Universal Robots PolyScope program: Simran_CNC_Program_FINAL.urp

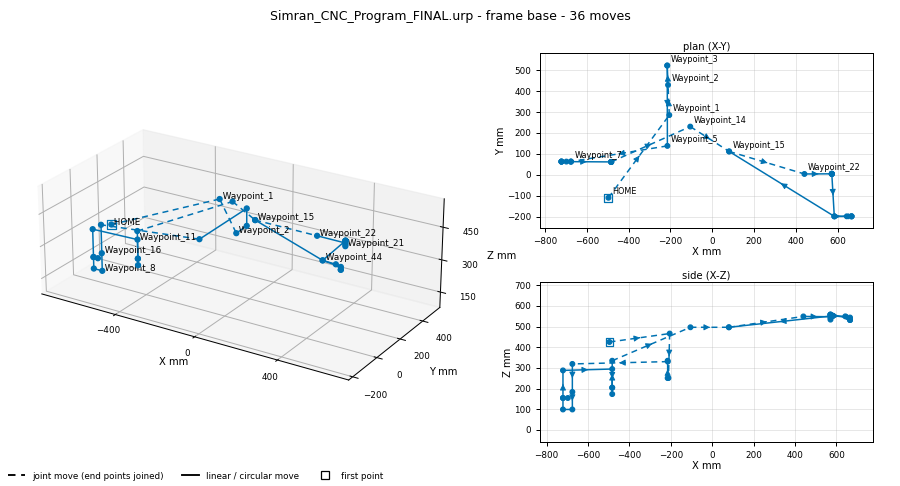
[picture p0: tool path of Simran_CNC_Program_FINAL.urp in frame base, 36 of 36 moves have a stored position in this frame; points joined in program order, loops and branches not executed]
Program Simran_CNC_Program_FINAL (createdIn=3.4.3.361 lastSavedIn=3.4.3.361 directory=/programs installation=default robotSerialNumber=2016352713)
Calibrated DH parameters: a=[0.000153, -0.131035, -0.301404, -0.000338, 0.000464, 0]; d=[0.089115, 288.344324, 295.555383, -583.78943, 0.09474, 0.082313]; alpha=[1.57022, 0.001403, 0.00043, 1.569471, -1.569661, 0]; deltaTheta=[-0.000066, 1.257544, -0.563043, -0.694494, -0.000004, 0.000038]
Robot Program (runOnlyOnce=true motionType=MoveJ speed=1.047198 acceleration=1.396263 useActiveTCP=false)
  MoveJ speed 60 deg/s, acceleration 80 deg/s^2 (useActiveTCP=false)
    Waypoint HOME: TCP in base x=-496.442 y=-110.074 z=425.318 mm, rx=1.2792 ry=2.857 rz=0.0029 rad; joints [-0.001, -88.582, 89.405, -90.126, -89.769, -41.695] deg
    Call Tool_OPEN
  'TURN TOWARDS CONVEYOR'
  MoveJ speed 60 deg/s, acceleration 80 deg/s^2 (useActiveTCP=false)
    Waypoint Waypoint_1: TCP in base x=-205.447 y=285.381 z=466.125 mm, rx=-1.2263 ry=-2.8909 rz=-0.0134 rad; joints [-72.357, -110.466, 101.648, -81.546, -90.206, -116.353] deg
  'PICK UP RAW MATERIALS BIN'
  MoveJ speed 60 deg/s, acceleration 80 deg/s^2 (useActiveTCP=false)
    Waypoint Waypoint_2: TCP in base x=-211.365 y=429.379 z=251.173 mm, rx=1.2208 ry=2.8789 rz=0.0239 rad; joints [-76.836, -86.876, 114.31, -117.592, -91.124, -120.798] deg
  MoveL speed 250 mm/s, acceleration 1200 mm/s^2 (useActiveTCP=false) feature=Base
    Waypoint Waypoint_3: TCP in base x=-215.251 y=522.375 z=251.019 mm, rx=1.2191 ry=2.8755 rz=0.0088 rad; joints [-78.664, -75.619, 100.862, -114.845, -90.993, -122.619] deg
    Waypoint Waypoint_4: motionParameters(jointSpeed=1.047198 jointAcceleration=1.396263 cartesianSpeed=0.02 cartesianAcceleration=0.02); TCP in base x=-215.258 y=522.371 z=334.743 mm, rx=1.2191 ry=2.8754 rz=0.0087 rad; joints [-78.665, -79.363, 92.558, -102.798, -90.989, -122.628] deg
    Waypoint Waypoint_5: TCP in base x=-214.547 y=138.032 z=330.506 mm, rx=1.2327 ry=2.8739 rz=0.0237 rad; joints [-57.762, -126.871, 129.262, -92.139, -91.154, -101.3] deg
  'PLACE RAW MATERIALS BIN'
  MoveJ speed 60 deg/s, acceleration 80 deg/s^2 (useActiveTCP=false)
    SuppressedNode
      Waypoint Waypoint_6: TCP in base x=-214.554 y=138.064 z=330.528 mm, rx=2.3465 ry=2.0595 rz=0.0117 rad; joints [-57.965, -126.737, 129.007, -91.172, -90.574, -50.482] deg
    Waypoint Waypoint_7: TCP in base x=-675.818 y=62.939 z=319.323 mm, rx=-2.9058 ry=-1.1583 rz=0.0302 rad; joints [-14.657, -63.822, 74.31, -101.769, -89.898, 31.98] deg
  MoveL speed 250 mm/s, acceleration 1200 mm/s^2 (useActiveTCP=false) feature=Base
    Waypoint Waypoint_16: TCP in base x=-675.802 y=62.877 z=183.922 mm, rx=-2.8969 ry=-1.1806 rz=0.0305 rad; joints [-14.658, -57.697, 85.778, -119.362, -89.886, 31.113] deg
    Waypoint Waypoint_8: motionParameters(jointSpeed=1.047198 jointAcceleration=1.396263 cartesianSpeed=0.02 cartesianAcceleration=0.02); TCP in base x=-675.776 y=62.901 z=99.21 mm, rx=-2.8958 ry=-1.1834 rz=0.0305 rad; joints [-14.66, -51.451, 89.635, -129.469, -89.886, 31.01] deg
    Waypoint Waypoint_9: TCP in base x=-721.173 y=62.9 z=99.19 mm, rx=-2.8958 ry=-1.1834 rz=0.0306 rad; joints [-13.746, -46.438, 80.218, -125.063, -89.908, 31.929] deg
    Waypoint Waypoint_10: motionParameters(jointSpeed=1.047198 jointAcceleration=1.396263 cartesianSpeed=0.25 cartesianAcceleration=1.2); TCP in base x=-721.174 y=62.931 z=154.677 mm, rx=-2.8958 ry=-1.1834 rz=0.0306 rad; joints [-13.745, -50.326, 77.932, -118.89, -89.901, 31.925] deg
    Waypoint Waypoint_17: motionParameters(jointSpeed=1.047198 jointAcceleration=1.396263 cartesianSpeed=0.02 cartesianAcceleration=0.02); TCP in base x=-697.665 y=62.978 z=154.655 mm, rx=-2.8959 ry=-1.1833 rz=0.0304 rad; joints [-14.203, -53.165, 82.942, -121.061, -89.89, 31.463] deg; flange x=-697.689 y=62.9 z=154.695 mm, rx=-2.8958 ry=-1.1834 rz=0.0306 rad
    Waypoint Waypoint_10: motionParameters(jointSpeed=1.047198 jointAcceleration=1.396263 cartesianSpeed=0.25 cartesianAcceleration=1.2); TCP in base x=-721.174 y=62.931 z=154.677 mm, rx=-2.8958 ry=-1.1834 rz=0.0306 rad; joints [-13.745, -50.326, 77.932, -118.89, -89.901, 31.925] deg
    Waypoint Waypoint_18: TCP in base x=-721.163 y=62.916 z=288.004 mm, rx=-2.8958 ry=-1.1834 rz=0.0304 rad; joints [-13.747, -56.577, 67.748, -102.456, -89.893, 31.91] deg; flange x=-721.174 y=62.931 z=288.056 mm, rx=-2.8958 ry=-1.1834 rz=0.0306 rad
  'PICK UP 1ST BLOCK'
  MoveL speed 250 mm/s, acceleration 1200 mm/s^2 (useActiveTCP=false) feature=Base
    Waypoint Waypoint_11: TCP in base x=-483.165 y=61.413 z=294.634 mm, rx=-2.894 ry=-1.1612 rz=-0.0146 rad; joints [-20.032, -88.315, 108.927, -111.051, -91.293, 26.31] deg; flange x=-483.17 y=61.41 z=294.731 mm, rx=-2.8939 ry=-1.1611 rz=-0.0143 rad
    Waypoint Waypoint_12: TCP in base x=-483.165 y=61.376 z=204.49 mm, rx=-2.8937 ry=-1.1612 rz=-0.0142 rad; joints [-20.033, -82.152, 117.078, -125.366, -91.297, 26.319] deg; flange x=-483.17 y=61.41 z=204.448 mm, rx=-2.8939 ry=-1.1611 rz=-0.0143 rad
    Waypoint Waypoint_23: motionParameters(jointSpeed=1.047198 jointAcceleration=1.396263 cartesianSpeed=0.02 cartesianAcceleration=0.02); TCP in base x=-483.17 y=61.41 z=173.567 mm, rx=-2.8939 ry=-1.1611 rz=-0.0143 rad; joints [-20.034, -79.281, 119.255, -130.412, -91.296, 26.321] deg
    Wait Sleep waitTime=0.5
    Call Tool_CLOSE
    Wait Sleep waitTime=1
    Waypoint Waypoint_12: motionParameters(jointSpeed=1.047198 jointAcceleration=1.396263 cartesianSpeed=0.02 cartesianAcceleration=0.02); TCP in base x=-483.165 y=61.376 z=204.49 mm, rx=-2.8937 ry=-1.1612 rz=-0.0142 rad; joints [-20.033, -82.152, 117.078, -125.366, -91.297, 26.319] deg; flange x=-483.17 y=61.41 z=204.448 mm, rx=-2.8939 ry=-1.1611 rz=-0.0143 rad
    Waypoint Waypoint_13: TCP in base x=-483.174 y=61.383 z=334.81 mm, rx=-2.894 ry=-1.1612 rz=-0.0146 rad; joints [-20.033, -90.016, 104.509, -104.919, -91.292, 26.304] deg
  MoveJ speed 60 deg/s, acceleration 80 deg/s^2 (useActiveTCP=false)
    Waypoint Waypoint_14: TCP in base x=-105.18 y=230.288 z=496.414 mm, rx=-1.2069 ry=-2.8666 rz=-0.0233 rad; joints [-91.595, -124.024, 103.951, -71.307, -88.599, -135.903] deg
    Waypoint Waypoint_15: TCP in base x=80.805 y=111.483 z=496.435 mm, rx=-1.2494 ry=-2.8485 rz=-0.0239 rad; joints [-180.178, -141.465, 106.176, -53.368, -88.466, -222.831] deg
    Wait Sleep waitTime=0.5
    Set DigitalOutput pin=door; digitalValue=1
    Wait Sleep waitTime=6
  'PLACE 1st BLOCK IN CNC'
  MoveJ speed 60 deg/s, acceleration 80 deg/s^2 (useActiveTCP=false)
    Waypoint Waypoint_22: TCP in base x=440.76 y=3.757 z=548.887 mm, rx=-1.2046 ry=-2.8864 rz=0.0111 rad; joints [-193.886, -95.387, 77.565, -71.268, -90.219, -238.54] deg
  MoveL speed 250 mm/s, acceleration 1200 mm/s^2 (useActiveTCP=false) feature=Base
    SuppressedNode
      Waypoint Waypoint_24: motionParameters(jointSpeed=1.047198 jointAcceleration=1.396263 cartesianSpeed=0.05 cartesianAcceleration=0.02); TCP in base x=551.7 y=-51.289 z=595.114 mm, rx=-2.8876 ry=-1.1713 rz=-0.0332 rad; joints [-197.055, -76.915, 50.59, -63.644, -88.035, -151.148] deg; flange x=551.728 y=-51.253 z=595.093 mm, rx=-2.8876 ry=-1.1713 rz=-0.0331 rad
    Waypoint Waypoint_20: motionParameters(jointSpeed=1.047198 jointAcceleration=1.396263 cartesianSpeed=0.05 cartesianAcceleration=0.025); TCP in base x=571.71 y=4.472 z=547.422 mm, rx=-1.2202 ry=-2.8799 rz=0.011 rad; joints [-190.617, -76.822, 57.791, -70.042, -90.155, -234.626] deg
    Waypoint Waypoint_21: motionParameters(jointSpeed=1.047198 jointAcceleration=1.396263 cartesianSpeed=0.05 cartesianAcceleration=0.01); TCP in base x=571.707 y=4.437 z=533.436 mm, rx=-1.2201 ry=-2.8798 rz=0.0111 rad; joints [-190.615, -77.492, 60.769, -72.35, -90.155, -234.624] deg; flange x=571.725 y=4.478 z=533.464 mm, rx=-1.2201 ry=-2.8799 rz=0.011 rad
    Call Tool_OPEN
    Wait Sleep waitTime=1
    Waypoint Waypoint_25: motionParameters(jointSpeed=1.047198 jointAcceleration=1.396263 cartesianSpeed=0.1 cartesianAcceleration=0.05); TCP in base x=571.711 y=4.432 z=557.354 mm, rx=-1.2201 ry=-2.8798 rz=0.0112 rad; joints [-190.623, -76.277, 55.552, -68.342, -90.155, -234.628] deg
    Call Tool_CLOSE
    Wait Sleep waitTime=1
    Waypoint Waypoint_26: motionParameters(jointSpeed=1.047198 jointAcceleration=1.396263 cartesianSpeed=0.25 cartesianAcceleration=0.1); TCP in base x=571.669 y=4.458 z=557.394 mm, rx=-0.0745 ry=-3.1304 rz=0.0184 rad; joints [-190.545, -76.378, 55.781, -68.858, -90.687, -277.744] deg; flange x=571.707 y=4.437 z=557.356 mm, rx=-0.0745 ry=-3.1303 rz=0.0184 rad
    SuppressedNode
      Waypoint Waypoint_27: motionParameters(jointSpeed=1.047198 jointAcceleration=1.396263 cartesianSpeed=0.025 cartesianAcceleration=0.01); TCP in base x=571.697 y=4.439 z=548.626 mm, rx=-0.0744 ry=-3.1304 rz=0.0184 rad; joints [-190.544, -76.857, 57.748, -70.346, -90.688, -277.743] deg
    SuppressedNode
      Waypoint Waypoint_26: motionParameters(jointSpeed=1.047198 jointAcceleration=1.396263 cartesianSpeed=0.1 cartesianAcceleration=0.05); TCP in base x=571.669 y=4.458 z=557.394 mm, rx=-0.0745 ry=-3.1304 rz=0.0184 rad; joints [-190.545, -76.378, 55.781, -68.858, -90.687, -277.744] deg; flange x=571.707 y=4.437 z=557.356 mm, rx=-0.0745 ry=-3.1303 rz=0.0184 rad
    Waypoint Waypoint_28: motionParameters(jointSpeed=1.047198 jointAcceleration=1.396263 cartesianSpeed=0.025 cartesianAcceleration=0.01); TCP in base x=571.706 y=4.422 z=540.796 mm, rx=-0.0745 ry=-3.1303 rz=0.0183 rad; joints [-190.543, -77.247, 59.44, -71.648, -90.688, -277.741] deg
    Waypoint Waypoint_26: motionParameters(jointSpeed=1.047198 jointAcceleration=1.396263 cartesianSpeed=0.25 cartesianAcceleration=0.1); TCP in base x=571.669 y=4.458 z=557.394 mm, rx=-0.0745 ry=-3.1304 rz=0.0184 rad; joints [-190.545, -76.378, 55.781, -68.858, -90.687, -277.744] deg; flange x=571.707 y=4.437 z=557.356 mm, rx=-0.0745 ry=-3.1303 rz=0.0184 rad
    Waypoint Waypoint_25: motionParameters(jointSpeed=1.047198 jointAcceleration=1.396263 cartesianSpeed=0.15 cartesianAcceleration=0.1); TCP in base x=571.711 y=4.432 z=557.354 mm, rx=-1.2201 ry=-2.8798 rz=0.0112 rad; joints [-190.623, -76.277, 55.552, -68.342, -90.155, -234.628] deg
    Waypoint Waypoint_44: motionParameters(jointSpeed=1.047198 jointAcceleration=1.396263 cartesianSpeed=0.1 cartesianAcceleration=0.05); TCP in base x=583.705 y=-198.923 z=551.901 mm, rx=-1.2205 ry=-2.8797 rz=0.0114 rad; joints [-209.035, -69.295, 47.056, -66.94, -90.423, -253.024] deg; flange x=583.758 y=-198.858 z=551.858 mm, rx=-1.2202 ry=-2.8797 rz=0.0112 rad
    Waypoint Waypoint_45: motionParameters(jointSpeed=1.047198 jointAcceleration=1.396263 cartesianSpeed=0.025 cartesianAcceleration=0.01); TCP in base x=643.414 y=-198.777 z=549.256 mm, rx=-1.2201 ry=-2.8799 rz=0.0113 rad; joints [-206.542, -58.298, 30.69, -61.552, -90.389, -250.524] deg; flange x=643.446 y=-198.824 z=549.179 mm, rx=-1.2201 ry=-2.8798 rz=0.0112 rad
    Waypoint Waypoint_46: motionParameters(jointSpeed=1.047198 jointAcceleration=1.396263 cartesianSpeed=0.025 cartesianAcceleration=0.01); TCP in base x=666.192 y=-198.791 z=531.433 mm, rx=-1.2198 ry=-2.8799 rz=0.0113 rad; joints [-205.699, -55.151, 28.355, -62.353, -90.381, -249.682] deg; flange x=666.19 y=-198.848 z=531.398 mm, rx=-1.2199 ry=-2.8798 rz=0.0112 rad
    Waypoint Waypoint_47: motionParameters(jointSpeed=1.047198 jointAcceleration=1.396263 cartesianSpeed=0.025 cartesianAcceleration=0.01); TCP in base x=666.173 y=-198.919 z=531.389 mm, rx=1.1834 ry=2.7931 rz=0.0671 rad; joints [-206.093, -58.682, 36.074, -73.343, -87.071, -249.923] deg; flange x=666.19 y=-198.848 z=531.398 mm, rx=1.1833 ry=2.7932 rz=0.0672 rad
    Waypoint Waypoint_48: motionParameters(jointSpeed=1.047198 jointAcceleration=1.396263 cartesianSpeed=0.025 cartesianAcceleration=0.01); TCP in base x=666.164 y=-198.888 z=543.546 mm, rx=-1.22 ry=-2.8797 rz=0.0113 rad; joints [-205.701, -53.361, 23.259, -59.048, -90.382, -249.683] deg
    Waypoint Waypoint_44: motionParameters(jointSpeed=1.047198 jointAcceleration=1.396263 cartesianSpeed=0.05 cartesianAcceleration=0.01); TCP in base x=583.705 y=-198.923 z=551.901 mm, rx=-1.2205 ry=-2.8797 rz=0.0114 rad; joints [-209.035, -69.295, 47.056, -66.94, -90.423, -253.024] deg; flange x=583.758 y=-198.858 z=551.858 mm, rx=-1.2202 ry=-2.8797 rz=0.0112 rad
    Waypoint Waypoint_15: motionParameters(jointSpeed=1.047198 jointAcceleration=1.396263 cartesianSpeed=0.25 cartesianAcceleration=0.1); TCP in base x=80.805 y=111.483 z=496.435 mm, rx=-1.2494 ry=-2.8485 rz=-0.0239 rad; joints [-180.178, -141.465, 106.176, -53.368, -88.466, -222.831] deg
    Wait Sleep waitTime=0.5
    Set DigitalOutput pin=door; digitalValue=0
    Wait Sleep waitTime=6
  'TOP TO BOTTOM'
  SuppressedNode
    MoveL speed 250 mm/s, acceleration 1200 mm/s^2 (useActiveTCP=false) feature=Base
      Set DigitalOutput pin=door; digitalValue=1
      Wait Sleep waitTime=6
      Waypoint Waypoint_22: motionParameters(jointSpeed=1.047198 jointAcceleration=1.396263 cartesianSpeed=0.25 cartesianAcceleration=0.1); TCP in base x=440.76 y=3.757 z=548.887 mm, rx=-1.2046 ry=-2.8864 rz=0.0111 rad; joints [-193.886, -95.387, 77.565, -71.268, -90.219, -238.54] deg
      Waypoint Waypoint_25: motionParameters(jointSpeed=1.047198 jointAcceleration=1.396263 cartesianSpeed=0.05 cartesianAcceleration=0.025); TCP in base x=571.711 y=4.432 z=557.354 mm, rx=-1.2201 ry=-2.8798 rz=0.0112 rad; joints [-190.623, -76.277, 55.552, -68.342, -90.155, -234.628] deg
      Call Tool_OPEN
      Wait Sleep waitTime=1
      Waypoint Waypoint_21: motionParameters(jointSpeed=1.047198 jointAcceleration=1.396263 cartesianSpeed=0.05 cartesianAcceleration=0.01); TCP in base x=571.707 y=4.437 z=533.436 mm, rx=-1.2201 ry=-2.8798 rz=0.0111 rad; joints [-190.615, -77.492, 60.769, -72.35, -90.155, -234.624] deg; flange x=571.725 y=4.478 z=533.464 mm, rx=-1.2201 ry=-2.8799 rz=0.011 rad
      Call Tool_CLOSE
      Wait Sleep waitTime=1
      Waypoint Waypoint_19: TCP in base x=571.698 y=4.439 z=560.42 mm, rx=-1.2202 ry=-2.8799 rz=0.0111 rad; joints [-190.62, -76.099, 54.845, -67.822, -90.153, -234.624] deg
      Waypoint Waypoint_24: TCP in base x=466.899 y=-34.446 z=560.48 mm, rx=-1.2202 ry=-2.8801 rz=0.011 rad; joints [-197.739, -91.133, 71.811, -69.799, -90.261, -241.762] deg
      Waypoint Waypoint_29: TCP in base x=332.54 y=-34.477 z=503.635 mm, rx=0.6252 ry=1.4734 rz=0.6267 rad; joints [-213.592, -111.621, 122.767, -191.492, -56.436, -223.787] deg
      Waypoint Waypoint_30: TCP in base x=413.921 y=-34.5 z=444.937 mm, rx=0.6252 ry=1.4734 rz=0.6267 rad; joints [-205.154, -95.603, 120.061, -204.763, -64.896, -223.835] deg
      Waypoint Waypoint_31: TCP in base x=413.908 y=-34.513 z=404.929 mm, rx=0.6253 ry=1.4734 rz=0.6266 rad; joints [-205.157, -92.629, 123.961, -211.635, -64.899, -223.839] deg
      Call Tool_OPEN
      Wait Sleep waitTime=1
      Waypoint Waypoint_32: motionParameters(jointSpeed=1.047198 jointAcceleration=1.396263 cartesianSpeed=0.05 cartesianAcceleration=0.01); TCP in base x=341.668 y=-34.501 z=404.92 mm, rx=0.6254 ry=1.4734 rz=0.6266 rad; joints [-212.365, -104.17, 133.396, -209.558, -57.68, -223.799] deg
      Waypoint Waypoint_33: motionParameters(jointSpeed=1.047198 jointAcceleration=1.396263 cartesianSpeed=0.05 cartesianAcceleration=0.01); TCP in base x=456.404 y=-34.465 z=589.86 mm, rx=-1.2203 ry=-2.88 rz=0.0107 rad; joints [-198.151, -91.019, 67.08, -65.184, -90.269, -242.178] deg
      Waypoint Waypoint_34: motionParameters(jointSpeed=1.047198 jointAcceleration=1.396263 cartesianSpeed=0.05 cartesianAcceleration=0.01); TCP in base x=565.728 y=-34.472 z=589.874 mm, rx=-1.2204 ry=-2.88 rz=0.0107 rad; joints [-194.649, -74.859, 48.544, -62.786, -90.203, -238.651] deg
      Waypoint Waypoint_35: motionParameters(jointSpeed=1.047198 jointAcceleration=1.396263 cartesianSpeed=0.05 cartesianAcceleration=0.01); TCP in base x=565.729 y=-34.449 z=574.404 mm, rx=-1.2202 ry=-2.88 rz=0.0106 rad; joints [-194.646, -75.994, 52.51, -65.617, -90.203, -238.649] deg
      Call Tool_CLOSE
      Wait Sleep waitTime=1
      Waypoint Waypoint_36: motionParameters(jointSpeed=1.047198 jointAcceleration=1.396263 cartesianSpeed=0.05 cartesianAcceleration=0.01); TCP in base x=565.735 y=-34.443 z=588.812 mm, rx=-1.2203 ry=-2.8801 rz=0.0107 rad; joints [-194.649, -74.944, 48.83, -62.987, -90.203, -238.651] deg
      Waypoint Waypoint_37: motionParameters(jointSpeed=1.047198 jointAcceleration=1.396263 cartesianSpeed=0.05 cartesianAcceleration=0.01); TCP in base x=378.265 y=-34.505 z=598.175 mm, rx=0.6269 ry=1.4775 rz=0.6256 rad; joints [-208.263, -105.692, 104.96, -179.298, -61.758, -223.949] deg
      Waypoint Waypoint_38: motionParameters(jointSpeed=1.047198 jointAcceleration=1.396263 cartesianSpeed=0.05 cartesianAcceleration=0.01); TCP in base x=382.478 y=-34.517 z=408.781 mm, rx=0.627 ry=1.4775 rz=0.6256 rad; joints [-207.853, -97.824, 127.848, -210.054, -62.197, -223.96] deg
      Waypoint Waypoint_39: motionParameters(jointSpeed=1.047198 jointAcceleration=1.396263 cartesianSpeed=0.025 cartesianAcceleration=0.01); TCP in base x=382.46 y=-34.495 z=390.09 mm, rx=0.6169 ry=1.454 rz=0.6313 rad; joints [-207.851, -95.528, 129.464, -215.6, -62.214, -223.196] deg
      Call Tool_OPEN
      Wait Sleep waitTime=1
      Waypoint Waypoint_40: motionParameters(jointSpeed=1.047198 jointAcceleration=1.396263 cartesianSpeed=0.05 cartesianAcceleration=0.01); TCP in base x=382.453 y=-34.53 z=561.181 mm, rx=0.617 ry=1.4539 rz=0.6314 rad; joints [-207.858, -104.454, 109.78, -186.993, -62.189, -223.19] deg
      Waypoint Waypoint_41: motionParameters(jointSpeed=1.047198 jointAcceleration=1.396263 cartesianSpeed=0.05 cartesianAcceleration=0.01); TCP in base x=548.004 y=-34.475 z=548.005 mm, rx=-1.2205 ry=-2.8802 rz=0.0109 rad; joints [-195.115, -80.211, 61.876, -70.777, -90.215, -239.117] deg; flange x=548.025 y=-34.482 z=547.959 mm, rx=-1.2204 ry=-2.8801 rz=0.0108 rad
      Call Tool_CLOSE
      Wait Sleep waitTime=1
      Waypoint Waypoint_42: motionParameters(jointSpeed=1.047198 jointAcceleration=1.396263 cartesianSpeed=0.05 cartesianAcceleration=0.01); TCP in base x=547.997 y=-34.458 z=556.525 mm, rx=-1.2203 ry=-2.8803 rz=0.0109 rad; joints [-195.116, -79.782, 60.04, -69.37, -90.215, -239.118] deg
      Waypoint Waypoint_43: motionParameters(jointSpeed=1.047198 jointAcceleration=1.396263 cartesianSpeed=0.05 cartesianAcceleration=0.01); TCP in base x=572.458 y=-72.283 z=556.569 mm, rx=-1.2205 ry=-2.8802 rz=0.0108 rad; joints [-198.148, -75.508, 54.714, -68.334, -90.257, -242.144] deg; flange x=572.504 y=-72.294 z=556.51 mm, rx=-1.2204 ry=-2.8801 rz=0.0108 rad
SubProgram -> Tool_OPEN
SubProgram -> Tool_CLOSE
SubProgram Tool_OPEN (keepSynchronizedWithDisk=false trackProgramExecution=false)
  Set DigitalOutput pin=digital_out[1]; digitalValue=1
  Set DigitalOutput pin=digital_out[0]; digitalValue=0
SubProgram Tool_CLOSE (keepSynchronizedWithDisk=false trackProgramExecution=false)
  Set DigitalOutput pin=digital_out[1]; digitalValue=0
  Set DigitalOutput (payload=0 tcpAsCog=true) pin=digital_out[0]; digitalValue=1
